{attribute 'GeneratedUsingTerminal: EJ4008-0000-0020'}
{attribute addProperty BoxType "EJ4008-0000-0020"}
{attribute addProperty Id "EtcSlaveTerminalBaseAO_Outputs_Channel_1AT %Q*AO_Outputs_Channel_BA7EBB7C2AO_Outputs_Channel_2AT %Q*AO_Outputs_Channel_BA7EBB7C2AO_Outputs_Channel_3AT %Q*AO_Outputs_Channel_BA7EBB7C2AO_Outputs_Channel_4AT %Q*AO_Outputs_Channel_BA7EBB7C2AO_Outputs_Channel_5AT %Q*AO_Outputs_Channel_BA7EBB7C2AO_Outputs_Channel_6AT %Q*AO_Outputs_Channel_BA7EBB7C2AO_Outputs_Channel_7AT %Q*AO_Outputs_Channel_BA7EBB7C2AO_Outputs_Channel_8AT %Q*AO_Outputs_Channel_BA7EBB7C2WcStateAT %I*WcState_0B2B16F91InfoDataAT %I*InfoData_32EB74EA10"}
{attribute addProperty CRC "3041722463"}
{attribute addProperty Size "27"}
TYPE EJ4008_B54D005F EXTENDS EtcSlaveTerminalBase :
STRUCT
	{attribute addProperty Name "AO_Outputs_Channel_1"}
	AO_Outputs_Channel_1 : AO_Outputs_Channel_BA7EBB7C;
	{attribute addProperty Name "AO_Outputs_Channel_2"}
	AO_Outputs_Channel_2 : AO_Outputs_Channel_BA7EBB7C;
	{attribute addProperty Name "AO_Outputs_Channel_3"}
	AO_Outputs_Channel_3 : AO_Outputs_Channel_BA7EBB7C;
	{attribute addProperty Name "AO_Outputs_Channel_4"}
	AO_Outputs_Channel_4 : AO_Outputs_Channel_BA7EBB7C;
	{attribute addProperty Name "AO_Outputs_Channel_5"}
	AO_Outputs_Channel_5 : AO_Outputs_Channel_BA7EBB7C;
	{attribute addProperty Name "AO_Outputs_Channel_6"}
	AO_Outputs_Channel_6 : AO_Outputs_Channel_BA7EBB7C;
	{attribute addProperty Name "AO_Outputs_Channel_7"}
	AO_Outputs_Channel_7 : AO_Outputs_Channel_BA7EBB7C;
	{attribute addProperty Name "AO_Outputs_Channel_8"}
	AO_Outputs_Channel_8 : AO_Outputs_Channel_BA7EBB7C;
	{attribute addProperty Name "WcState"}
	WcState : WcState_0B2B16F9;
	{attribute addProperty Name "InfoData"}
	InfoData : InfoData_32EB74EA;
END_STRUCT
END_TYPE

(* stored: Version 1.2.0.0, ProductVersion 3.1.4024.9
   DUT EJ4008_B54D005F: Id {d991424a-37f3-4968-a8f5-600399b4e89a} *)
